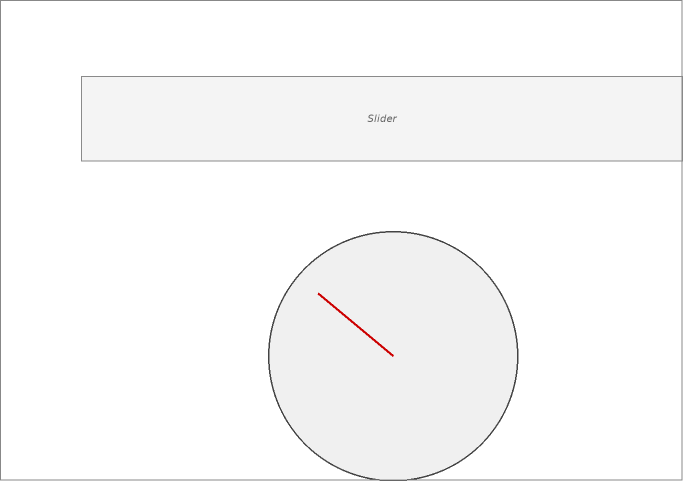
VISUALIZATION Visualization  // 683x481
    Slider (81,76 602x85), variable: MAIN.nRawAnalogInput, scale 0..32767
    Meter360 (268,231 250x250), value: MAIN.fMotorSpeedPercent, style: Meter-Meter360-Gray, scale format: %.1f, scale 0..100
END_VISUALIZATION

(* stored: Version 1.1.0.1
   Visu Visualization: Id {3caf9944-a084-49ec-b4c4-d785b250beb7} *)
